// TIA Portal project "babu_ConveyorWithDelay" (V15)

(* hardware
DEVICE "S7-1200 station_1"  S7-1200 Station
   slot 0: "Rack_0"  S7-1200 Rack  Rack  V1.0
   slot 1: "PLC_1"  CPU 1212C DC/DC/DC  6ES7 212-1AE40-0XB0  V4.2
*)

// ===== PLC "PLC_1"  CPU 1212C DC/DC/DC =====

VAR_GLOBAL   // PLC tag table "Default tag table"
   "START PUSH BUTTON" AT %M0.0 : Bool;
   "START PBM" AT %M0.1 : Bool;
   "STOP PUSH BUTTON" AT %M0.2 : Bool;
   "STOP PBM" AT %M0.3 : Bool;
   "CONVEYOR" AT %Q0.0 : Bool;
   "STOP DELAY" AT %M0.4 : Bool;
   "SIGNAL LIGHT" AT %Q0.1 : Bool;
END_VAR

// folder: System blocks/Program resources

DATA_BLOCK "IEC_Timer_0_DB"   // DB1
{ S7_Optimized_Access := 'TRUE' }
AUTHOR : Simatic
FAMILY : IEC
NAME : IEC_TMR
VERSION : 1.0
// stored: InstanceOfName IEC_TIMER
"IEC_TIMER"
BEGIN
END_DATA_BLOCK

DATA_BLOCK "IEC_Timer_0_DB_1"   // DB2
{ S7_Optimized_Access := 'TRUE' }
AUTHOR : Simatic
FAMILY : IEC
NAME : IEC_TMR
VERSION : 1.0
// stored: InstanceOfName IEC_TIMER
"IEC_TIMER"
BEGIN
END_DATA_BLOCK

DATA_BLOCK "IEC_Timer_0_DB_2"   // DB3
{ S7_Optimized_Access := 'TRUE' }
AUTHOR : Simatic
FAMILY : IEC
NAME : IEC_TMR
VERSION : 1.0
// stored: InstanceOfName IEC_TIMER
"IEC_TIMER"
BEGIN
END_DATA_BLOCK

// folder: (top level)

ORGANIZATION_BLOCK "Main"   // OB1, LAD, ProgramCycle
TITLE = "Main Program Sweep (Cycle)"
{ S7_Optimized_Access := 'TRUE' }
VERSION : 0.1
   VAR_INPUT
      Initial_Call : Bool;   // Initial call of this OB
      Remanence : Bool;   // =True, if remanent data are available
   END_VAR
BEGIN

REGION Network 1
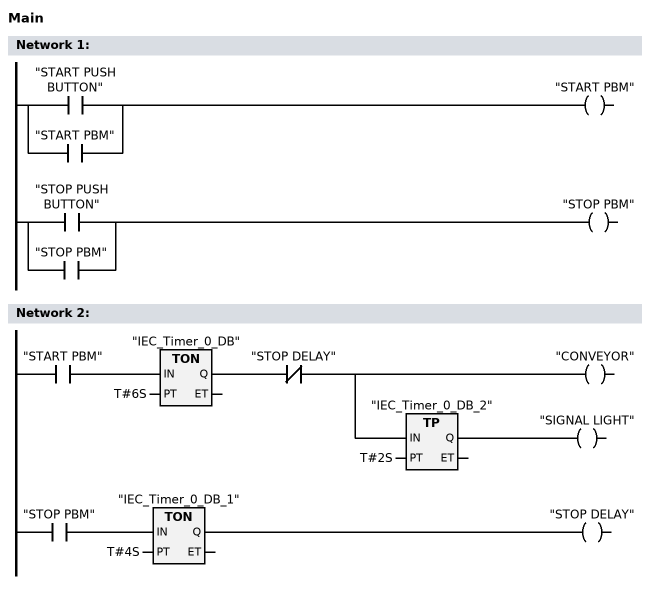
   RUNG wire#powerrail
      Contact( "START PUSH BUTTON" )
      wire#w1
      Coil( "START PBM" )
   END_RUNG
   RUNG wire#powerrail
      Contact( "START PBM" )
   END_RUNG wire#w1
   RUNG wire#powerrail
      Contact( "STOP PUSH BUTTON" )
      wire#w2
      Coil( "STOP PBM" )
   END_RUNG
   RUNG wire#powerrail
      Contact( "STOP PBM" )
   END_RUNG wire#w2
   // the same network as SCL:
   "START PBM" := "START PUSH BUTTON" OR "START PBM";
   "STOP PBM" := "STOP PUSH BUTTON" OR "STOP PBM";
END_REGION

REGION Network 2
   "IEC_Timer_0_DB".TON(IN := "START PBM", PT := T#6S);
   "CONVEYOR" := "IEC_Timer_0_DB".Q AND NOT "STOP DELAY";
   "IEC_Timer_0_DB_2".TP(IN := "CONVEYOR", PT := T#2S);
   "SIGNAL LIGHT" := "IEC_Timer_0_DB_2".Q;
   "IEC_Timer_0_DB_1".TON(IN := "STOP PBM", PT := T#4S);
   "STOP DELAY" := "IEC_Timer_0_DB_1".Q;
END_REGION
END_ORGANIZATION_BLOCK